PROGRAM pouReadHMIMessages
VAR


	openfile: FB_FILEOPEN;
	closefile: FB_FileClose;
	
	startOpeningFile: BOOL;

	OpenedFileNum: UINT;
	startRead: BOOL;
	startClosingfile: BOOL;
END_VAR

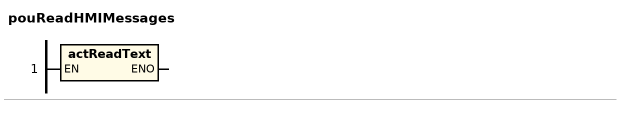
// NETWORK 1
actReadText();

ACTION actReadText:



IF startRead THEN
	
	//self clear for 1 scan
	startRead:= FALSE;
	
	startOpeningFile := TRUE;
					
END_IF

//open file
openfile	(sNetId:=,
			sPathName:='C:\PLC\Messages\Mc_Alarms.XML',
			nMode:=FOPEN_MODEREAD,
			ePath:=PATH_GENERIC,
			bExecute:=startOpeningFile,
			tTimeout:=T#1S
			);
startOpeningFile := FALSE;		

//do something else here to read more of the file in
OpenedFileNum := openfile.hFile;


IF OpenedFileNum = 0 THEN
	startClosingfile:=TRUE;
END_IF


//close the file when read in the XML data
closefile	(sNetId:=,
			hFile:= OpenedFileNum,
			bExecute:=startClosingfile,
			tTimeout:=T#1S
			);
startClosingfile:=FALSE;
END_ACTION

END_PROGRAM

(* stored: Version 1.1.0.1, ProductVersion 3.1.4024.12
   POU pouReadHMIMessages: Id {ce838f3d-32dc-4330-919e-70024cdd9543}, SpecialFunc None
   Action actReadText: Id {ef7559f8-d0a7-4bd6-9ac5-587f43038718} *)
